// TIA Portal V19 export
DATA_BLOCK "DATE_AND_TIME"   // DB5
{ S7_Optimized_Access := 'FALSE' }
   VAR
      SET_YEAR : DWord;
      SET_MONTH : DWord;
      SET_DAY : DWord;
      SET_HOUR : DWord;
      SET_MIN : DWord;
      SET_SEC : DWord;
   END_VAR
BEGIN
END_DATA_BLOCK
